(* CODESYS project PLC.project
   Title: PLC
   Version: 0.0.0.0
   Author: Oleksandr

Project tree, tasks and I/O mapping:
  Controller : TM241CEC24T/U, Schneider Electric, order no. TM241CEC24T/U, version 4.0.6.18
    application Application
      task MAST (cyclic, interval 20 ms, priority 15, watchdog 100 ms x 1) calls Main
      global variables GVL
      program Main [ST]
    DQ : Digital Outputs, Schneider Electric, version 4.0.6.18
        output qwDQ_QW0 : WORD  // QW0
        output qbDQ_QB1 : BYTE  // QB1
    Counters : Counters, Schneider Electric, version 4.0.6.18
    Pulse_Generators : Pulse Generators, Schneider Electric, version 4.0.6.18
    Cartridge_1 : Cartridge, Schneider Electric, version 4.0.6.18
    IO_Bus : IO bus - TM3, Schneider Electric, version 4.0.6.18
      Module_4 : TM3AQ4/G, Schneider Electric, order no. TM3AQ4/G, version 1.0.0.12
          output qiModule_4_QW0 : INT  // QW0
          output qiModule_4_QW1 : INT  // QW1
          output qiModule_4_QW2 : INT  // QW2
          output qiModule_4_QW3 : INT  // QW3
          input  ibModule_4_IBStatusQW0 : BYTE  // IBStatusQW0
          input  ibModule_4_IBStatusQW1 : BYTE  // IBStatusQW1
          input  ibModule_4_IBStatusQW2 : BYTE  // IBStatusQW2
          input  ibModule_4_IBStatusQW3 : BYTE  // IBStatusQW3
      Module_6 : TM3AI8/G, Schneider Electric, order no. TM3AI8/G, version 1.0.0.17
          input  iiModule_6_IW0 : INT  // IW0
          input  iiModule_6_IW1 : INT  // IW1
          input  iiModule_6_IW2 : INT  // IW2
          input  iiModule_6_IW3 : INT  // IW3
          input  iiModule_6_IW4 : INT  // IW4
          input  iiModule_6_IW5 : INT  // IW5
          input  iiModule_6_IW6 : INT  // IW6
          input  iiModule_6_IW7 : INT  // IW7
          input  ibModule_6_IBStatusIW0 : BYTE  // IBStatusIW0
          input  ibModule_6_IBStatusIW1 : BYTE  // IBStatusIW1
          input  ibModule_6_IBStatusIW2 : BYTE  // IBStatusIW2
          input  ibModule_6_IBStatusIW3 : BYTE  // IBStatusIW3
          input  ibModule_6_IBStatusIW4 : BYTE  // IBStatusIW4
          input  ibModule_6_IBStatusIW5 : BYTE  // IBStatusIW5
          input  ibModule_6_IBStatusIW6 : BYTE  // IBStatusIW6
          input  ibModule_6_IBStatusIW7 : BYTE  // IBStatusIW7
      Module_1 : TM3DQ8R/G, Schneider Electric, order no. TM3DQ8R/G, version 1.0.1.4
          output qbModule_1_QB0 : BYTE  // QB0
    COM_Bus : COM bus, Schneider Electric, version 4.0.6.18
    DI : Digital Inputs, Schneider Electric, version 4.0.6.18
        input  iwDI_IW0 : WORD  // IW0
        input  ibDI_IB1 : BYTE  // IB1
    Ethernet_1 : Ethernet Network, Schneider Electric, version 4.0.6.18
    Serial_Line_1 : Serial line, Schneider Electric, version 4.0.6.18
      SoMachine_Network_Manager : SoMachine-Network Manager, Schneider Electric, version 4.0.0.2
    Serial_Line_2 : Serial line, Schneider Electric, version 4.0.6.18
      Modbus_Manager : Modbus Manager, Schneider Electric, version 4.0.0.2
    CAN_1 : CANopen bus, Schneider Electric, version 4.0.6.18
*)

// Controller/Application/GVL
VAR_GLOBAL
	QX3_0 AT %QX3.0:BOOL;
	QX3_1 AT %QX3.1:BOOL;
	QX3_2 AT %QX3.2:BOOL;
	QX3_3 AT %QX3.3:BOOL;
	QX3_4 AT %QX3.4:BOOL;
	QX3_5 AT %QX3.5:BOOL;
	QX3_6 AT %QX3.6:BOOL;
	QX3_7 AT %QX3.7:BOOL;
	QX4_0 AT %QX4.0:BOOL;
	QX4_1 AT %QX4.1:BOOL;
	QX4_2 AT %QX4.2:BOOL;
	QX4_3 AT %QX4.3:BOOL;
	QX4_4 AT %QX4.4:BOOL;
	QX4_5 AT %QX4.5:BOOL;
	QX4_6 AT %QX4.6:BOOL;
	QX4_7 AT %QX4.7:BOOL;
	
	M0_5:BOOL; //AUTO-HAND Switch
END_VAR

VAR_GLOBAL RETAIN
	MW0 AT %MW0:WORD;
	MW4 AT %MW4:WORD;
END_VAR

// Controller/Application/Main
PROGRAM Main
VAR
	WORD_AS_BIT_1: WORD_AS_BIT;
	WORD_AS_BIT_0: WORD_AS_BIT;
END_VAR

WORD_AS_BIT_0( W:= MW0,B05=> M0_5);
WORD_AS_BIT_1( W:= MW4,B01=> QX3_0, B02=> QX3_1, B03=> QX3_2, B04=> QX3_3, B05=> QX3_4, B07=> QX3_5, B08=> QX3_6, B09=> QX3_7, B10=> QX4_0, B11=> QX4_1, B12=> QX4_2, B13=> QX4_3);

END_PROGRAM
